FUNCTION_BLOCK RelativeMOVE
VAR_INPUT
	MoveAxisIdx			: INT;
	MoveDistance		: LREAL;
	MoveVelocity			: LREAL;
	MoveAcceleration		: LREAL;
	MoveDeceleration		: LREAL;
	MoveJerk			: LREAL;
END_VAR
VAR_OUTPUT
END_VAR
VAR
END_VAR


Axis[MoveAxisIdx].fbMC_MoveRelative[1](
	Execute  		:= TRUE,
	Distance		:= MoveDistance,
	Velocity  		:= MoveVelocity,
	Acceleration   := MoveAcceleration,
	Deceleration  := MoveDeceleration,
	Jerk			:= MoveJerk,
	BufferMode     := MC_BlendingHigh,
	Axis			:= Axis[MoveAxisIdx].Axis
);

Axis[MoveAxisIdx].fbMC_MoveRelative[1](
	Execute  		:= FALSE,
	Axis			:= Axis[MoveAxisIdx].Axis
);

END_FUNCTION_BLOCK

(* stored: Version 1.1.0.1, ProductVersion 3.1.4024.9
   POU RelativeMOVE: Id {fc080483-2f9d-4e38-b8d6-84dde55fc444}, SpecialFunc None *)
